// SIMATIC STEP 7 (V5.x) project day3
// CPU: CPU 315-2 DP
// CPU: CPU 315-2 DP
// station: Hardware
// station: SIMATIC 300(1)
// station: P_ADR_BUS
// station: P_ADR_BUS
// station: Hardware
// station: SIMATIC 300(2)
// program: S7 Program(1)
// program: S7 Program(3)

SYMBOL_TABLE
"START_BUTTON"	I 0.0	BOOL
"STOP_BUTTON"	I 0.1	BOOL
"STOP_COIL"	M 0.0	BOOL
"STOP_BIT"	M 0.1	BOOL
"MOTOR1"	Q 4.0	BOOL
"MOTOR2"	Q 4.1	BOOL
"LAMP"	Q 4.2	BOOL
"MOTOR_1_TIMER"	T 0	TIMER
"MOTOR_2_TIMER"	T 1	TIMER
END_SYMBOL_TABLE

ORGANIZATION_BLOCK OB 1
TITLE = "Main Program Sweep (Cycle)"
VERSION : 0.1
VAR_TEMP
  OB1_EV_CLASS : BYTE ;	//Bits 0-3 = 1 (Coming event), Bits 4-7 = 1 (Event class 1)
  OB1_SCAN_1 : BYTE ;	//1 (Cold restart scan 1 of OB 1), 3 (Scan 2-n of OB 1)
  OB1_PRIORITY : BYTE ;	//Priority of OB Execution
  OB1_OB_NUMBR : BYTE ;	//1 (Organization block 1, OB1)
  OB1_RESERVED_1 : BYTE ;	//Reserved for system
  OB1_RESERVED_2 : BYTE ;	//Reserved for system
  OB1_PREV_CYCLE : INT ;	//Cycle time of previous OB1 scan (milliseconds)
  OB1_MIN_CYCLE : INT ;	//Minimum cycle time of OB1 (milliseconds)
  OB1_MAX_CYCLE : INT ;	//Maximum cycle time of OB1 (milliseconds)
  OB1_DATE_TIME : DATE_AND_TIME ;	//Date and time OB1 started
END_VAR
BEGIN
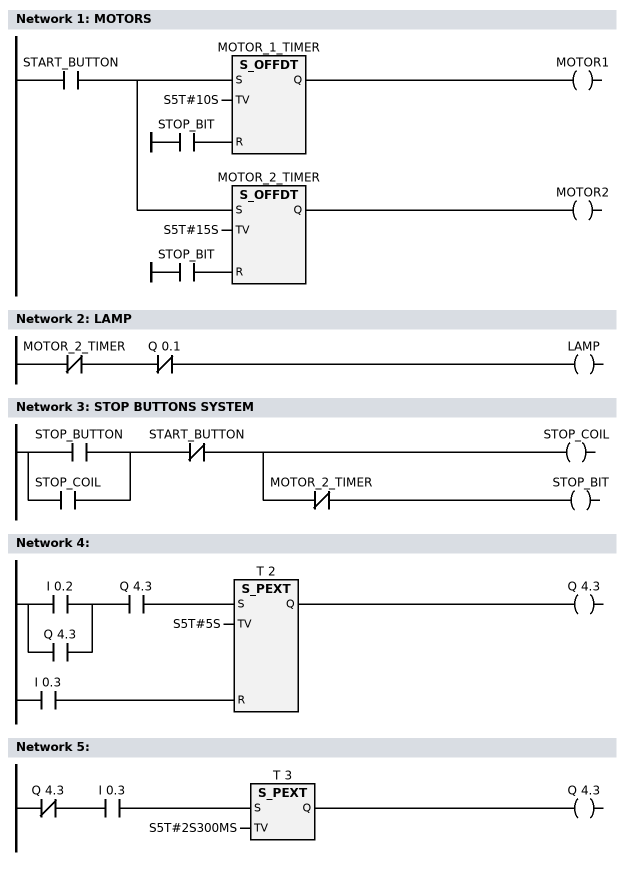
NETWORK
TITLE = MOTORS
      A     "START_BUTTON";
      =     L 20.0;
      A     L 20.0;
      L     S5T#10S;
      SF    "MOTOR_1_TIMER";
      A     "STOP_BIT";
      R     "MOTOR_1_TIMER";
      NOP   0;
      NOP   0;
      A     "MOTOR_1_TIMER";
      =     "MOTOR1";
      A     L 20.0;
      L     S5T#15S;
      SF    "MOTOR_2_TIMER";
      A     "STOP_BIT";
      R     "MOTOR_2_TIMER";
      NOP   0;
      NOP   0;
      A     "MOTOR_2_TIMER";
      =     "MOTOR2";
NETWORK
TITLE = LAMP
      AN    "MOTOR_2_TIMER";
      AN    Q 0.1;
      =     "LAMP";
NETWORK
TITLE = STOP BUTTONS SYSTEM
      A(;
      O     "STOP_BUTTON";
      O     "STOP_COIL";
      );
      AN    "START_BUTTON";
      =     L 20.0;
      A     L 20.0;
      BLD   102;
      =     "STOP_COIL";
      A     L 20.0;
      AN    "MOTOR_2_TIMER";
      =     "STOP_BIT";
NETWORK
TITLE =
      A(;
      O     I 0.2;
      O     Q 4.3;
      );
      A     Q 4.3;
      L     S5T#5S;
      SE    T 2;
      A     I 0.3;
      R     T 2;
      NOP   0;
      NOP   0;
      A     T 2;
      =     Q 4.3;
NETWORK
TITLE =
      AN    Q 4.3;
      A     I 0.3;
      L     S5T#2S300MS;
      SE    T 3;
      NOP   0;
      NOP   0;
      NOP   0;
      A     T 3;
      =     Q 4.3;
END_ORGANIZATION_BLOCK

ORGANIZATION_BLOCK OB 1
VERSION : 0.1
BEGIN
// (block stored without names or comments; labels and parameter names are numbered)
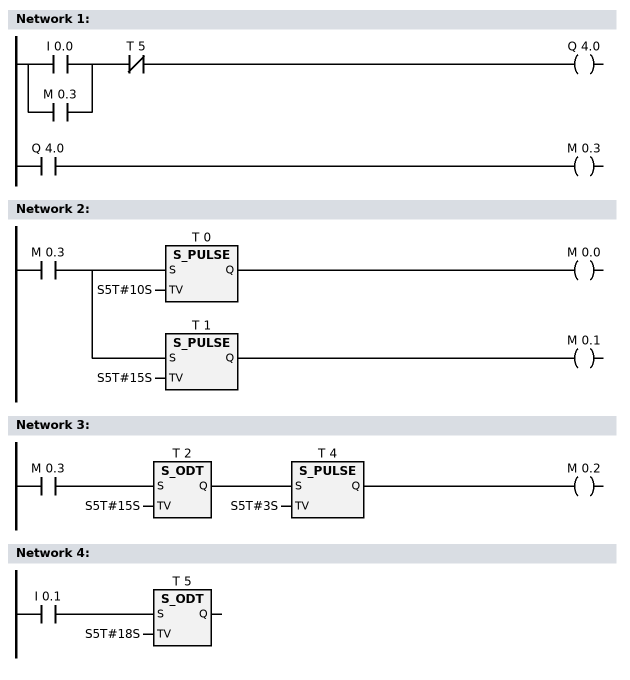
NETWORK
TITLE =
      A(;
      O     I 0.0;
      O     M 0.3;
      );
      AN    T 5;
      =     Q 4.0;
      A     Q 4.0;
      =     M 0.3;
NETWORK
TITLE =
      A     M 0.3;
      =     L 20.0;
      A     L 20.0;
      L     S5T#10S;
      SP    T 0;
      NOP   0;
      NOP   0;
      NOP   0;
      A     T 0;
      =     M 0.0;
      A     L 20.0;
      L     S5T#15S;
      SP    T 1;
      NOP   0;
      NOP   0;
      NOP   0;
      A     T 1;
      =     M 0.1;
NETWORK
TITLE =
      A(;
      A     M 0.3;
      L     S5T#15S;
      SD    T 2;
      NOP   0;
      NOP   0;
      NOP   0;
      A     T 2;
      );
      L     S5T#3S;
      SP    T 4;
      NOP   0;
      NOP   0;
      NOP   0;
      A     T 4;
      =     M 0.2;
NETWORK
TITLE =
      A     I 0.1;
      L     S5T#18S;
      SD    T 5;
      NOP   0;
      NOP   0;
      NOP   0;
      NOP   0;
END_ORGANIZATION_BLOCK
